FUNCTION_BLOCK OutfeedModule EXTENDS FB_PackML_BaseModule
VAR
	testComplete : BOOL;
END_VAR

// This method serves as the entry point for all underlying FB logic
METHOD PUBLIC CyclicLogic

// This method should be called cyclically by descendant function blocks by invoking SUPER^.CyclicLogic().  Alternatively, the contents of this method could be reimplemented entirely in which case a call to this method would not be necessary.
IF NOT _InitComplete THEN
	_InitComplete := Initialize();
	RETURN;
END_IF

SUPER^.CyclicLogic();

//
IF testComplete THEN
	testComplete := FALSE;
	Trace('Outfeed changing state to Complete');
	ChangeState(State := E_PMLCommand.Complete);
END_IF
END_METHOD

// Basic module initialization logic
METHOD PROTECTED Initialize : BOOL;

// This method is called by CyclicLogic() as required
Initialize := FALSE;
CASE DescendantSequenceState OF
	0:
		//Setup Config
		_LogModeChanges			:= FALSE;
		_LogStateChanges		:= FALSE;
		DescendantSequenceState := DescendantSequenceState + 10;

	10: // Call the Super 
		IF SUPER^.Initialize() THEN
			Initialize := TRUE;
		END_IF
END_CASE
END_METHOD

END_FUNCTION_BLOCK

(* stored: Version 1.1.0.1, ProductVersion 3.1.4026.12
   POU OutfeedModule: Id {217672e2-776d-43db-a4bd-00471447b980}, SpecialFunc None
   Method CyclicLogic: Id {71472b5c-82e4-4981-b631-e99c50fd0cc2}
   Method Initialize: Id {1814c178-8629-4868-8222-3c7807509b08} *)
